Staubli VAL3: page_viewPallet.pjx

--- page_viewPallet.pjx ---
Parameters version=s7.2.1 stackSize=5000 millimeterUnit=true
Program file=buildList.pgx
Program file=listAdd.pgx
Program file=loadPage.pgx
Program file=main.pgx
Program file=makeMaxSizeList.pgx
Program file=onEnterEvent.pgx
Program file=onExit.pgx
Program file=onF1Event.pgx
Program file=onF2Event.pgx
Program file=onF3Event.pgx
Program file=onF4Event.pgx
Program file=onF5Event.pgx
Program file=onF6Event.pgx
Program file=onF7Event.pgx
Program file=onF8Event.pgx
Program file=onStart.pgx
Program file=refresh.pgx
Program file=refreshDynamic.pgx
Program file=refreshStatic.pgx
Data file=page_viewPallet.dtx
Library alias=page path=Disk://kernel/template/page/page.pjx
Library alias=use path=Disk://kernel/userPage/userPage.pjx
Library alias=language2 path=Disk://trajectory/PALLET/language/language.pjx
Library alias=pallet path=Disk://trajectory/PALLET/PALLET.pjx
Library alias=saveData path=Disk://saveData/saveData.pjx
Library alias=language path=Disk://kernel/language/language.pjx
Library alias=cycleStatus path=Disk://cycleStatus/cycleStatus.pjx
Library alias=OnEvent path=Disk://OnEvent/OnEvent.pjx

--- page_viewPallet.dtx ---
num nIndex
num nKey
num nMax
num nRefresh
num nTime = 2
num nView
string sEvent
public string sItems
string sList
string sMenu
string sMessage
string sPalletName
bool bButton[8]
bool bLarge
bool bOnActionLine
frame fView = {fatherId=world[0]}
pointRx pOrigin = {wrist=wfree, fatherId=fView[0]}
pointRx pPoints[4]
  [0] = {wrist=wfree, fatherId=world[0]}
  [1] = {wrist=wfree, fatherId=world[0]}
  [2] = {wrist=wfree, fatherId=world[0]}
  [3] = {wrist=wfree, fatherId=world[0]}

--- main.pgx ---
public program main()
  local bool l_bSave
begin
  // INIT
  call onStart()
  // LOOP UNTIL nKey=255
  do
    call refresh()
    nKey=getKey()
    call use:listevent(nKey,nIndex,sEvent)
    nView=use:nView
    if nIndex>=0
      switch nKey
        case 259
          // TAB
          bLarge=!bLarge
          call use:setView(bLarge)
        break
        case 271
          // RESET ALL
          call onF1Event()
        break
        case 272
          // edit traj
          call onF2Event()
        break
        case 273
          call onF3Event()
        break
        case 274
          call onF4Event()
        break
        case 275
        break
        case 276
          // back
          call onF6Event(sPalletName[nIndex])
        break
        case 277
          // next
          call onF7Event(sPalletName[nIndex])
        break
        case 278
          // reset
          call onF8Event(sPalletName[nIndex])
        break
        case 270
          call onEnterEvent(sPalletName[nIndex])
        break
      endSwitch
    endIf
    // release
    delay(0)
  until nKey==255
  // on Exit
  call onExit()
end

--- buildList.pgx ---
program buildList()
  local num i
  local string l_sPalletName
  local num l_nPosition[4]
  local string l_sEmpty
  local num l_nSize
begin
  // INIT the list
  l_sEmpty=""
  call use:stringCopy(l_sEmpty,sList)
  //
  // Build the list
  //
  for i=0 to size(sPalletName)-1
    // scan all
    if sPalletName[i]!=""
      l_sPalletName=sPalletName[i]
      call pallet:getPalletPos(l_sPalletName,l_nPosition)
      call pallet:getSizePallet(l_sPalletName,l_nSize)
      call use:strfill(l_sPalletName,12,l_sPalletName)
      call listAdd(l_sPalletName+"> "+toString("",l_nPosition+1)+"/"+toString("",l_nSize))
    endIf
  endFor
  // refresh it
  // rebuild the list
  call use:listempty()
  call use:listadd(sList)
end

--- listAdd.pgx ---
program listAdd(string x_sEvent)
begin
  // add in the queue
  if sList!=""
    insert(sList[size(sList)])
  endIf
  sList[size(sList)-1]=x_sEvent
end

--- loadPage.pgx ---
program loadPage(string x_sPage, string& x_sItems[])
// load the next page
  local num i
begin
  // look if the page libload is correct
  i=page:libLoad(x_sPage)
  delay(0)
  logMsg("[KERNEL] INTERFACE:PAGE LIBLOAD "+x_sPage+" result "+toString("",i))
  if i!=0
    popUpMsg("Loading page "+x_sPage+" error CODE "+toString("",i))
  else
    // copy all the field from x_sItems to the next page
    call use:stringCopy(x_sItems,page:sItems)
    call page:main()
    // to give back
    call use:stringCopy(page:sItems,x_sItems)
  endIf
end

--- makeMaxSizeList.pgx ---
program makeMaxSizeList(num& x_nResult[])
  local string l_sPalletName
  local num l_nSize
  local num i
  local num l_nSizePallet[4]
  local string l_sTemp
  local string l_sEmpty
begin
  //
  // INIT
  //
  sPalletName=""
  // make the list of the max size list of pallet
  call pallet:getSize(l_nSize)
  resize(sPalletName,1,max(1,l_nSize))
  resize(nMax,1,max(1,l_nSize))
  //
  // build the list
  //
  for i=0 to l_nSize-1
    call pallet:get(l_sPalletName,i)
    if l_sPalletName!=""
      call pallet:getSizePallet(l_sPalletName,l_nSizePallet)
      nMax[i]=l_nSizePallet
      sPalletName[i]=l_sPalletName
    endIf
  endFor
end

--- onEnterEvent.pgx ---
program onEnterEvent(string x_sName)
  local num l_nSize[4]
  local num i
  local string l_sProg
  local num l_nIndex
  local num l_nPosition[4]
  local string l_sEmpty
begin
  //
  // NB sEvent is the selected
  // element in the LIST
  //
  call pallet:getPalletPos(x_sName,l_nPosition)
  call pallet:getSizePallet(x_sName,l_nSize)
  //
  if nIndex>=0
    i=find(sEvent,">")+1
  endIf
  //
  // clean the line
  call use:listcursor(use:nView,false)
  //
  if l_nSize>1
    // absolute
    l_sEmpty=""
    l_nPosition=l_nPosition+1
    call use:changeValue(l_nPosition,1,l_nSize,i+40-use:nBottomX,use:nView+1,l_sEmpty)
    call pallet:setPalletPos(x_sName,l_nPosition-1)
    // refresh it
    call buildList()
  endIf
  use:bUseRefresh=true
end

--- onExit.pgx ---
program onExit()
begin
end

--- onF1Event.pgx ---
program onF1Event()
  local string l_sPalletName
  local num i
begin
  // look if the bButton is enable
  if bButton[0]
    call pallet:reset()
  endIf
end

--- onF2Event.pgx ---
program onF2Event()
  local string l_sPath
  local string l_sItems[2]
begin
  // look if the bButton is enable
  if bButton[1]
    //
  endIf
end

--- onF5Event.pgx ---
program onF5Event(bool& x_bSave[])
begin
  // look if the bButton is enable
  if bButton[4]
    //
  endIf
end

--- onF6Event.pgx ---
program onF6Event(string x_sName)
begin
  // look if the bButton is enable
  if bButton[5]
    // RESET
    call pallet:setPalletPos(x_sName,0)
    // refresh it
    call buildList()
    use:bUseRefresh=true
  endIf
end

--- onF7Event.pgx ---
program onF7Event(string x_sName)
  local num l_nMax
begin
  // look if the bButton is enable
  if bButton[6]
    // BACK
    call pallet:back(x_sName)
    // refresh it
    call buildList()
    use:bUseRefresh=true
  endIf
end

--- onF8Event.pgx ---
program onF8Event(string x_sName)
begin
  // look if the bButton is enable
  if bButton[7]
    // NEXT
    call pallet:next(x_sName)
    // refresh it
    call buildList()
    use:bUseRefresh=true
  endIf
end

--- onStart.pgx ---
program onStart()
  local num i
  local num l_nResult
  local string l_sPath
  local string l_sMessage
begin
  // language
  //
  call language2:getLanguage(l_sPath)
  if l_sPath!=language2:libPath()+"/"+saveData:language
    // set language
    call language2:setLanguage(language2:libPath()+"/"+saveData:language)
  endIf
  // logMsg
  logMsg("[KERNEL] INTERFACE:PAGE VIEW ALL PALLET")
  // reset the Key pressure
  call use:nullKey(nKey)
  call language:message(l_sMessage,19)
  call use:timerDialog(l_sMessage,0)
  // make the max_size of all
  call makeMaxSizeList(l_nResult)
  if l_nResult==0
    //
    call buildList()
    // build the page
    call refreshStatic()
    // define the list
  else
    call language:message(l_sMessage,-7)
    popUpMsg(l_sMessage+" ; "+toString("",l_nResult))
    logMsg("[KERNEL] INTERFACE:ERROR LOADING VIEW PALLET ERROR CODE "+toString("",l_nResult))
  endIf
end

--- refreshDynamic.pgx ---
program refreshDynamic()
begin
  // DO NOT CHANGE
  nRefresh=clock()
  use:bUseRefresh=false
  //
  // ADD HERE
  //
  call buildList()
  //
  // refresh the cursor
  use:nView=nView
  // refresh the list
  call use:listupdate(nIndex-nView)
end

--- refreshStatic.pgx ---
program refreshStatic()
  local string l_sMenu
begin
  cls()
  //
  // set the view of the page..
  //
  // SET THE PAGE NUMBER
  use:nPage=100
  // USE <>PROFILE for <>PAGE
  use:nPage=use:nPage+abs(limit(saveData:mode,0,2)-2)
  // SET THE VIEW OF THE PAGE
  call language2:page(l_sMenu,use:nPage)
  // define the menu
  call use:stringToArray(l_sMenu,sMenu)
  //
  call use:setMenu(sMenu,true,3)
  call use:getMenu(sMenu,bButton)
  //
  // CREATE THE LIST
  //
  // define your list size for default
  call use:setSizeList(19,0,19,11)
  call use:setView(bLarge)
  //
  call use:listcreate("")
  //
end
